SYSTEM Test Delay Chain
  (* Version 1.0, 2005-06-24, Goran, Chalmers *)
  DEVICE Test Device : DeviceType_not_used
    RESOURCE TestResource : ResourceType_not_used
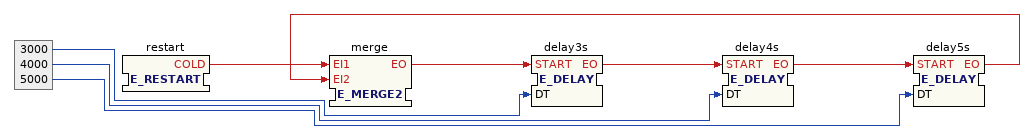
      FBS
        restart : E_RESTART;
        merge : E_MERGE2;
        delay3s : E_DELAY;
        delay4s : E_DELAY;
        delay5s : E_DELAY;
      END_FBS
      EVENT_CONNECTIONS
        restart.COLD TO merge.EI1;
        merge.EO TO delay3s.START;
        delay3s.EO TO delay4s.START;
        delay4s.EO TO delay5s.START;
        delay5s.EO TO merge.EI2;
      END_CONNECTIONS
      DATA_CONNECTIONS
        3000 TO delay3s.DT;
        4000 TO delay4s.DT;
        5000 TO delay5s.DT;
      END_CONNECTIONS
    END_RESOURCE
  END_DEVICE
END_SYSTEM
